INTERFACE I_SessionHeaderAccessor

METHOD PUBLIC TryGetSessionIdFromRequest : BOOL
VAR_INPUT
	Request : I_Request;
	Destination : REFERENCE TO T_MAXSTRING;
END_VAR
END_METHOD

METHOD PUBLIC UpdateRequestWithSessionId
VAR_INPUT
	Request : I_Request;
	SessionId : T_MAXSTRING;
END_VAR
END_METHOD

METHOD PUBLIC UpdateResponseWithSessionId
VAR_INPUT
	Response : I_ServerResponse;
	SessionId : T_MAXSTRING;
END_VAR
END_METHOD

END_INTERFACE

(* stored: Version 1.1.0.1, ProductVersion 3.1.4024.12
   Itf I_SessionHeaderAccessor: Id {2d1dce30-eb78-0293-331d-481e9066be23}
   Method TryGetSessionIdFromRequest: Id {9d51c638-f9ed-08e2-2323-78794f6e0d82}
   Method UpdateRequestWithSessionId: Id {e6801f14-5d46-0a10-1b69-078e5cf73e75}
   Method UpdateResponseWithSessionId: Id {132ddb2b-519c-020a-351b-92159d5a1957} *)
